FUNCTION_BLOCK ReleaseMaster
VAR_INPUT
	bReleaseAckIn : BOOL;
END_VAR

VAR_OUTPUT
	bSetRelease : BOOL;
	bLastHandshakeSuccesful : BOOL;
END_VAR


VAR
	fbReleaseAckInEvent : R_TRIG;
	fbSetReleaseEvent : R_TRIG;
	fbHandshakeSuccessfulEvent : R_TRIG;
END_VAR

fbReleaseAckInEvent(CLK:=bReleaseAckIn);
fbSetReleaseEvent(CLK:=bSetRelease);

IF fbReleaseAckInEvent.Q
THEN
	OnReleaseAckIn();
END_IF

IF fbSetReleaseEvent.Q
THEN
	OnSetRelease();
END_IF

IF fbHandshakeSuccessfulEvent.Q
THEN	
	bLastHandshakeSuccesful := TRUE;
END_IF

METHOD OnHandshakeSuccessful : BOOL
VAR_INPUT
END_VAR
END_METHOD

METHOD OnReleaseAckIn : BOOL
VAR_INPUT
END_VAR
bSetRelease := FALSE;
END_METHOD

METHOD OnSetRelease : BOOL
VAR_INPUT
END_VAR
bLastHandshakeSuccesful := FALSE;
END_METHOD

METHOD SetReleaseClient : BOOL
VAR_IN_OUT
	fbReleaseClient : ReleaseClient;
END_VAR
bReleaseAckIn := fbReleaseClient.bReleaseAckOut;
fbReleaseClient.bReleasePresent := bSetRelease;

fbHandshakeSuccessfulEvent(CLK:=fbReleaseClient.bLastHandshakeSuccesful);
END_METHOD

END_FUNCTION_BLOCK

(* stored: Version 1.1.0.1, ProductVersion 3.1.4024.2
   POU ReleaseMaster: Id {1bd31e51-9896-4100-ac8e-9b92f3d9fa3e}, SpecialFunc None
   Method OnHandshakeSuccessful: Id {551f9349-6943-4e72-9ef9-62337d0d7078}
   Method OnReleaseAckIn: Id {c21cbb55-3370-4b71-9b4c-c79118c49480}
   Method OnSetRelease: Id {3b73cf21-3105-42af-b778-25ce8d80ca5f}
   Method SetReleaseClient: Id {3c12957f-715b-46b2-a40b-55310a207da0} *)
